# B&R Automation Studio project ChoiceBagging_SSBP (part 2)

#### Error.ld - Error detected
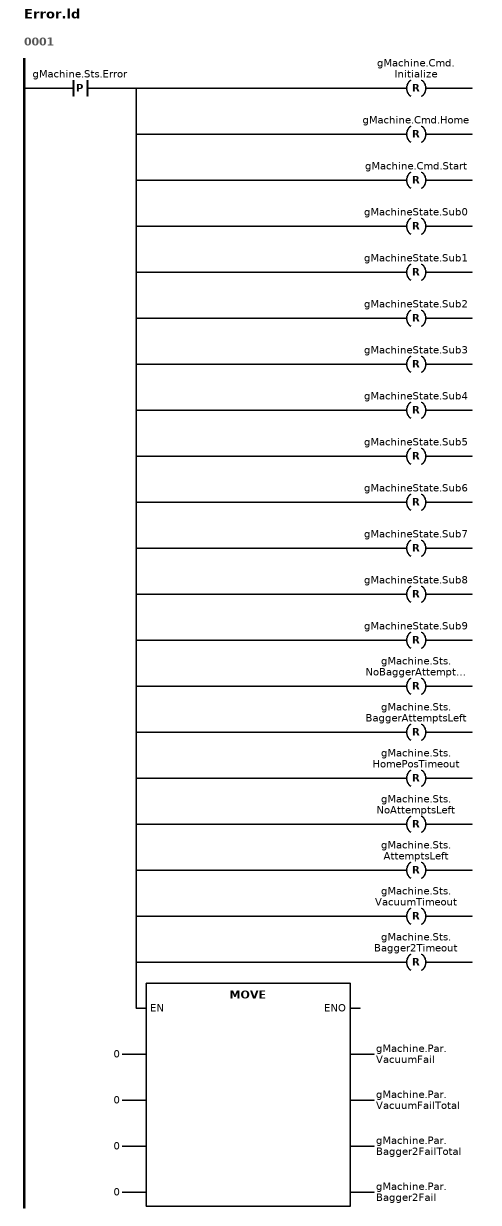
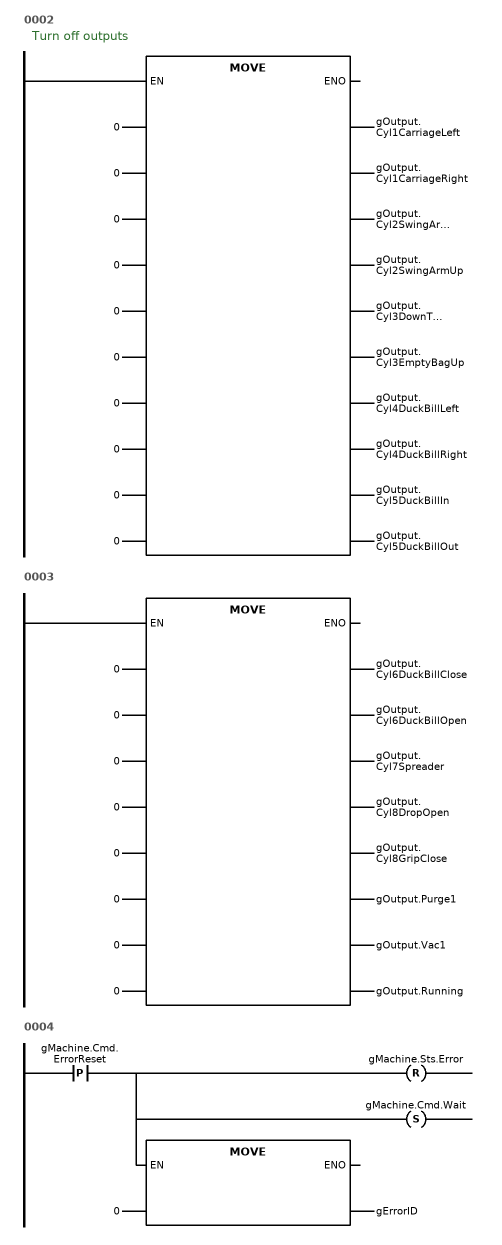
Ladder, written as Structured Text:
```iecst
ACTION Error:
VAR
    _e1 : R_TRIG;
    _e2 : R_TRIG;
END_VAR
(* Network 1 *)
_e1(CLK := gMachine.Sts.Error);
IF _e1.Q THEN
    gMachine.Cmd.Initialize := FALSE;
    gMachine.Cmd.Home := FALSE;
    gMachine.Cmd.Start := FALSE;
    gMachineState.Sub0 := FALSE;
    gMachineState.Sub1 := FALSE;
    gMachineState.Sub2 := FALSE;
    gMachineState.Sub3 := FALSE;
    gMachineState.Sub4 := FALSE;
    gMachineState.Sub5 := FALSE;
    gMachineState.Sub6 := FALSE;
    gMachineState.Sub7 := FALSE;
    gMachineState.Sub8 := FALSE;
    gMachineState.Sub9 := FALSE;
    gMachine.Sts.NoBaggerAttemptsLeft := FALSE;
    gMachine.Sts.BaggerAttemptsLeft := FALSE;
    gMachine.Sts.HomePosTimeout := FALSE;
    gMachine.Sts.NoAttemptsLeft := FALSE;
    gMachine.Sts.AttemptsLeft := FALSE;
    gMachine.Sts.VacuumTimeout := FALSE;
    gMachine.Sts.Bagger2Timeout := FALSE;
    gMachine.Par.VacuumFail := 0;
    gMachine.Par.VacuumFailTotal := 0;
    gMachine.Par.Bagger2FailTotal := 0;
    gMachine.Par.Bagger2Fail := 0;
END_IF;

(* Network 2: Turn off outputs *)
gOutput.Cyl1CarriageLeft := 0;
gOutput.Cyl1CarriageRight := 0;
gOutput.Cyl2SwingArmDown := 0;
gOutput.Cyl2SwingArmUp := 0;
gOutput.Cyl3DownToEmptyBag := 0;
gOutput.Cyl3EmptyBagUp := 0;
gOutput.Cyl4DuckBillLeft := 0;
gOutput.Cyl4DuckBillRight := 0;
gOutput.Cyl5DuckBillIn := 0;
gOutput.Cyl5DuckBillOut := 0;

(* Network 3 *)
gOutput.Cyl6DuckBillClose := 0;
gOutput.Cyl6DuckBillOpen := 0;
gOutput.Cyl7Spreader := 0;
gOutput.Cyl8DropOpen := 0;
gOutput.Cyl8GripClose := 0;
gOutput.Purge1 := 0;
gOutput.Vac1 := 0;
gOutput.Running := 0;

(* Network 4 *)
_e2(CLK := gMachine.Cmd.ErrorReset);
IF _e2.Q THEN
    gMachine.Sts.Error := FALSE;
    gMachine.Cmd.Wait := TRUE;
    gErrorID := 0;
END_IF;
END_ACTION
```

#### Wait.ld -  Waiting
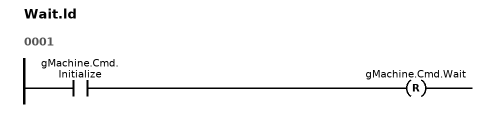
Ladder, written as Structured Text:
```iecst
ACTION Wait:
(* Network 1 *)
IF gMachine.Cmd.Initialize THEN gMachine.Cmd.Wait := FALSE; END_IF;
END_ACTION
```

#### Pause.ld - Pause / resume
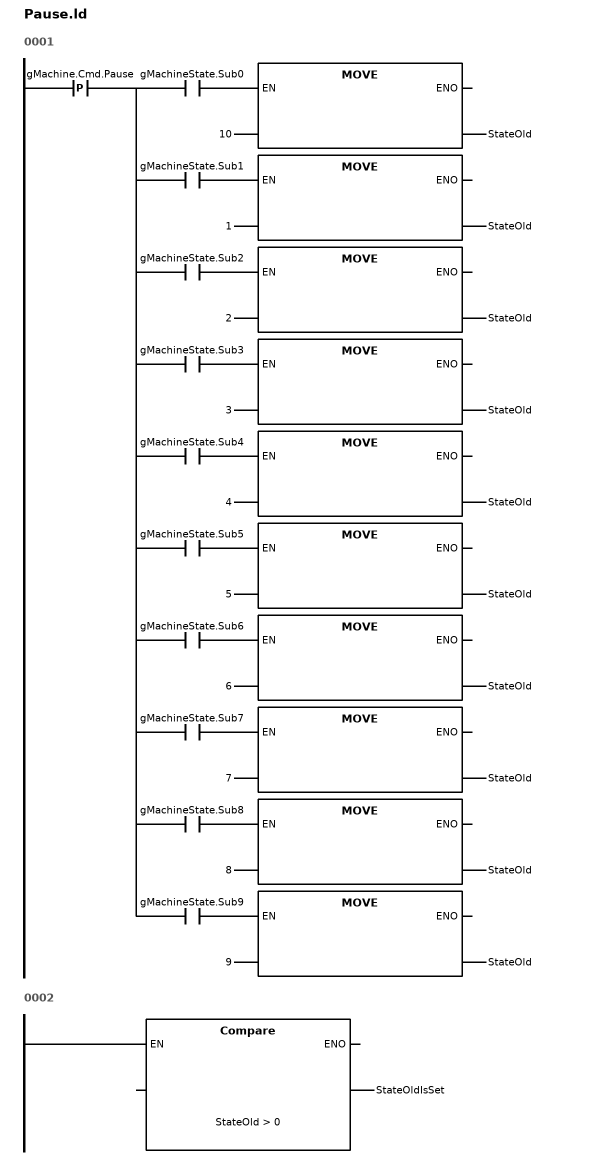
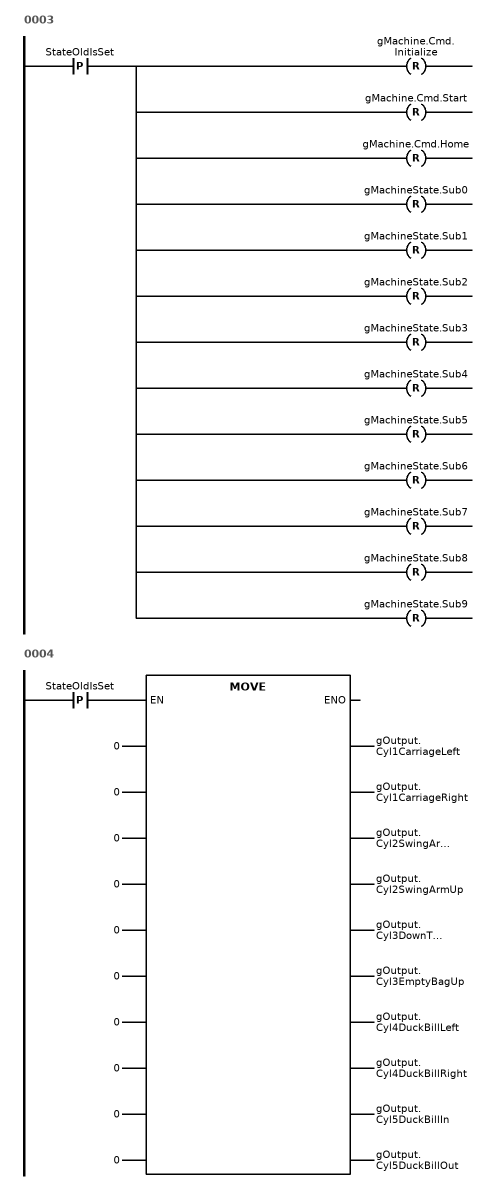
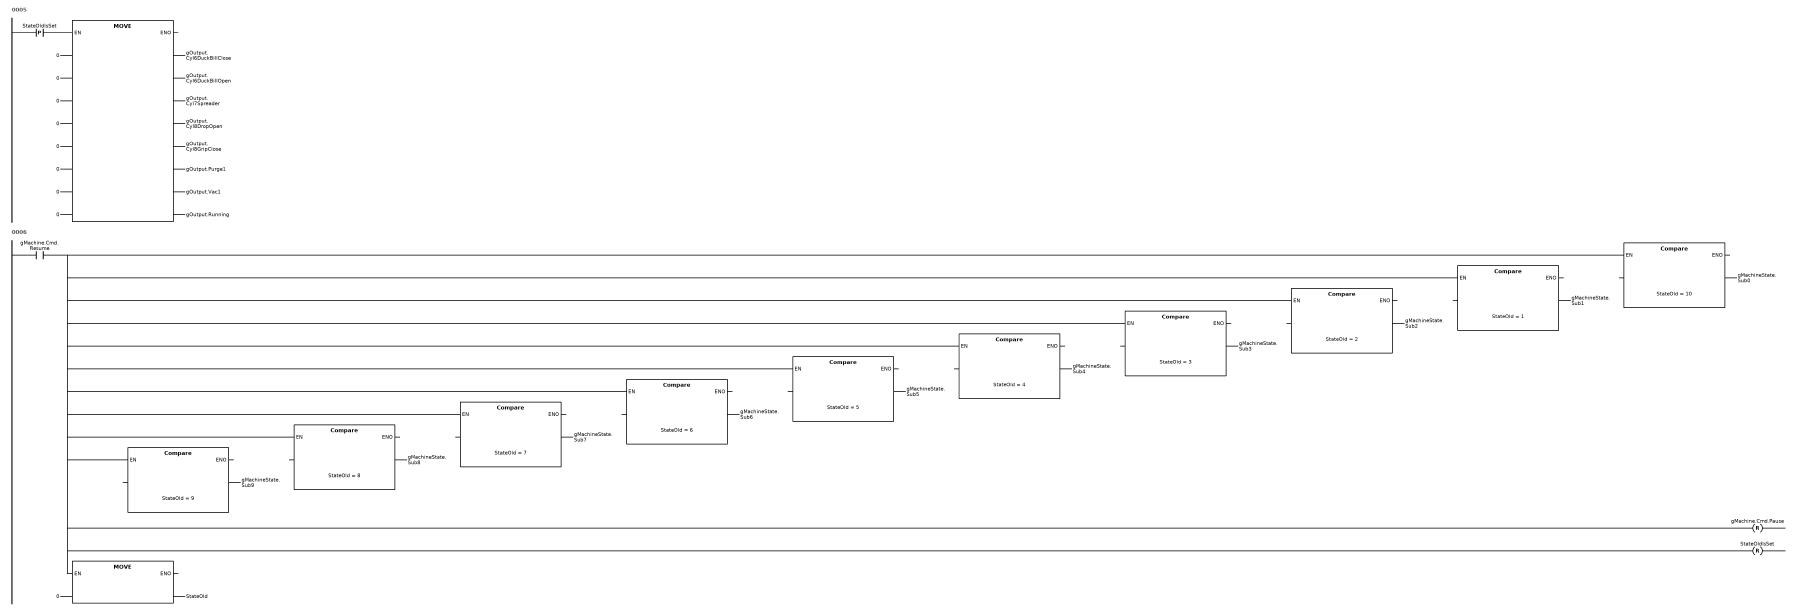
Ladder, written as Structured Text:
```iecst
ACTION Pause:
VAR
    _e1 : R_TRIG;
    _e2 : R_TRIG;
    _e3 : R_TRIG;
    _e4 : R_TRIG;
    _p5 : BOOL;
END_VAR
(* Network 1 *)
_e1(CLK := gMachine.Cmd.Pause);
IF _e1.Q AND gMachineState.Sub0 THEN StateOld := 10; END_IF;
IF _e1.Q AND gMachineState.Sub1 THEN StateOld := 1; END_IF;
IF _e1.Q AND gMachineState.Sub2 THEN StateOld := 2; END_IF;
IF _e1.Q AND gMachineState.Sub3 THEN StateOld := 3; END_IF;
IF _e1.Q AND gMachineState.Sub4 THEN StateOld := 4; END_IF;
IF _e1.Q AND gMachineState.Sub5 THEN StateOld := 5; END_IF;
IF _e1.Q AND gMachineState.Sub6 THEN StateOld := 6; END_IF;
IF _e1.Q AND gMachineState.Sub7 THEN StateOld := 7; END_IF;
IF _e1.Q AND gMachineState.Sub8 THEN StateOld := 8; END_IF;
IF _e1.Q AND gMachineState.Sub9 THEN StateOld := 9; END_IF;

(* Network 2 *)
StateOldIsSet := StateOld > 0;

(* Network 3 *)
_e2(CLK := StateOldIsSet);
IF _e2.Q THEN
    gMachine.Cmd.Initialize := FALSE;
    gMachine.Cmd.Start := FALSE;
    gMachine.Cmd.Home := FALSE;
    gMachineState.Sub0 := FALSE;
    gMachineState.Sub1 := FALSE;
    gMachineState.Sub2 := FALSE;
    gMachineState.Sub3 := FALSE;
    gMachineState.Sub4 := FALSE;
    gMachineState.Sub5 := FALSE;
    gMachineState.Sub6 := FALSE;
    gMachineState.Sub7 := FALSE;
    gMachineState.Sub8 := FALSE;
    gMachineState.Sub9 := FALSE;
END_IF;

(* Network 4 *)
_e3(CLK := StateOldIsSet);
IF _e3.Q THEN
    gOutput.Cyl1CarriageLeft := 0;
    gOutput.Cyl1CarriageRight := 0;
    gOutput.Cyl2SwingArmDown := 0;
    gOutput.Cyl2SwingArmUp := 0;
    gOutput.Cyl3DownToEmptyBag := 0;
    gOutput.Cyl3EmptyBagUp := 0;
    gOutput.Cyl4DuckBillLeft := 0;
    gOutput.Cyl4DuckBillRight := 0;
    gOutput.Cyl5DuckBillIn := 0;
    gOutput.Cyl5DuckBillOut := 0;
END_IF;

(* Network 5 *)
_e4(CLK := StateOldIsSet);
IF _e4.Q THEN
    gOutput.Cyl6DuckBillClose := 0;
    gOutput.Cyl6DuckBillOpen := 0;
    gOutput.Cyl7Spreader := 0;
    gOutput.Cyl8DropOpen := 0;
    gOutput.Cyl8GripClose := 0;
    gOutput.Purge1 := 0;
    gOutput.Vac1 := 0;
    gOutput.Running := 0;
END_IF;

(* Network 6 *)
IF gMachine.Cmd.Resume THEN
    gMachineState.Sub0 := StateOld = 10;
    gMachineState.Sub1 := StateOld = 1;
    gMachineState.Sub2 := StateOld = 2;
    gMachineState.Sub3 := StateOld = 3;
    gMachineState.Sub4 := StateOld = 4;
    gMachineState.Sub5 := StateOld = 5;
    gMachineState.Sub6 := StateOld = 6;
    gMachineState.Sub7 := StateOld = 7;
    gMachineState.Sub8 := StateOld = 8;
    gMachineState.Sub9 := StateOld = 9;
END_IF;
_p5 := gMachine.Cmd.Resume;
IF gMachine.Cmd.Resume THEN gMachine.Cmd.Pause := FALSE; END_IF;
IF _p5 THEN
    StateOldIsSet := FALSE;
    StateOld := 0;
END_IF;
END_ACTION
```

### Program Logical/AlarmCtrl (IEC)

#### Cyclic.ld - Cyclic code
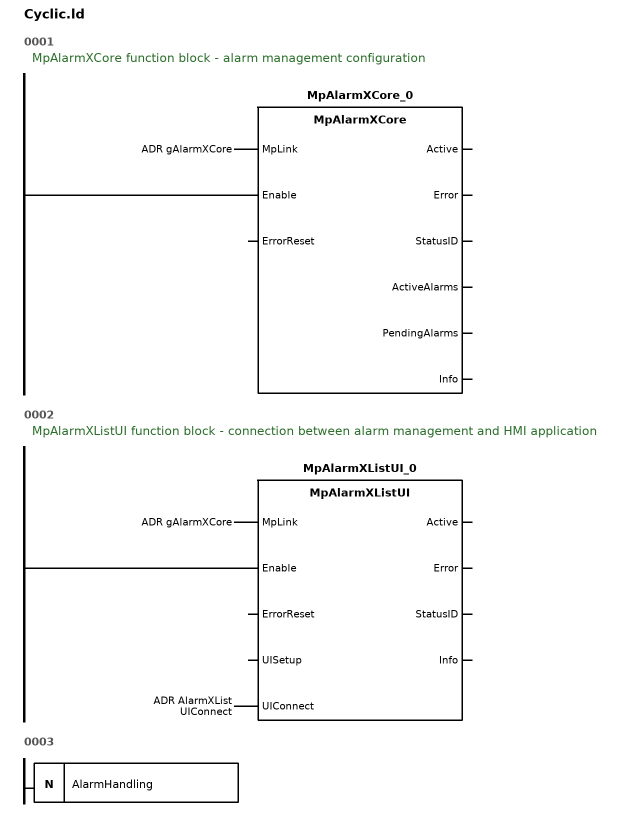
Ladder, written as Structured Text:
```iecst
(*********************************************************************************
 * Copyright: 	Hartfiel Automation
 * Author:    	cashley
 * Created:   	August 5, 2019/2:01 PM
 * Description: This file contains the control logic for handling the alarm system.
 *********************************************************************************)
 PROGRAM _CYCLIC
(* Network 1: MpAlarmXCore function block - alarm management configuration *)
MpAlarmXCore_0(MpLink := ADR(gAlarmXCore), Enable := TRUE);

(* Network 2: MpAlarmXListUI function block - connection between alarm management and HMI application *)
MpAlarmXListUI_0(MpLink := ADR(gAlarmXCore), Enable := TRUE, UIConnect := ADR(AlarmXListUIConnect));

(* Network 3 *)
AlarmHandling;
END_PROGRAM
```

#### Variables.var - Local variables
```iecst
VAR
	MpAlarmXCore_0 : MpAlarmXCore; (*Function block for MpAlarmXCore*)
	MpAlarmXListUI_0 : MpAlarmXListUI; (*Function block for MpAlarmXListUI*)
	AlarmXListUIConnect : MpAlarmXListUIConnectType; (*MpAlarmXListUIConnect type*)
	ErrorString : STRING[255]; (*String for MpAlarmXSet unique alarm code*)
END_VAR
```

#### AlarmHandling.st - Alarm handling
```iecst
ACTION AlarmHandling:

	//Error ID determines unique name for MpAlarmXSet
	IF gErrorID = HOMING_TIMEOUT THEN
		ErrorString := 'HomingTimeout';
	ELSIF gErrorID = SAFE_TO_RUN THEN
		ErrorString := 'SafetyStatus';
	ELSIF gErrorID = CONVEYOR THEN
		ErrorString := 'ConveyorStatus';
	ELSIF gErrorID = MODULE_OK THEN
		ErrorString := 'ModuleStatus';
	ELSIF gErrorID = VACUUM_FAILURE THEN
		ErrorString := 'VacuumFailure';
	ELSIF gErrorID = BAG_ON_SPOUT_FAILURE THEN
		ErrorString := 'Bagger2Failure';
	END_IF

	//MpAlarmXSet - enables user-defined alarms
	IF EDGEPOS(gMachine.Sts.Error) THEN
		MpAlarmXSet(MpLink := gAlarmXCore, Name := ErrorString);
	END_IF

	//Error acknowledge and reset
	IF gMachine.Sts.Error = FALSE THEN
		gMachine.Cmd.ErrorReset := FALSE;
	END_IF

END_ACTION
```

### Program Logical/IOCtrl (IEC)

#### Cyclic.ld
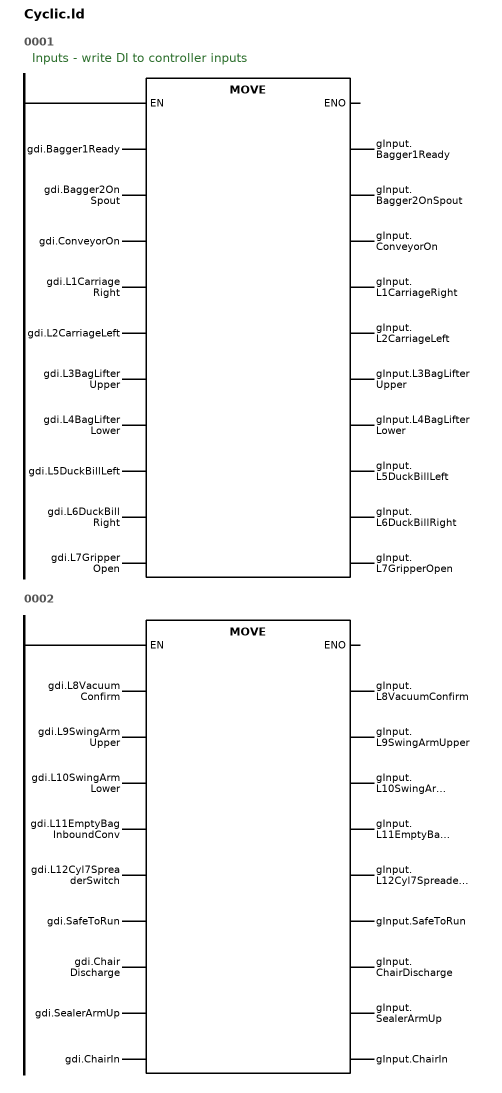
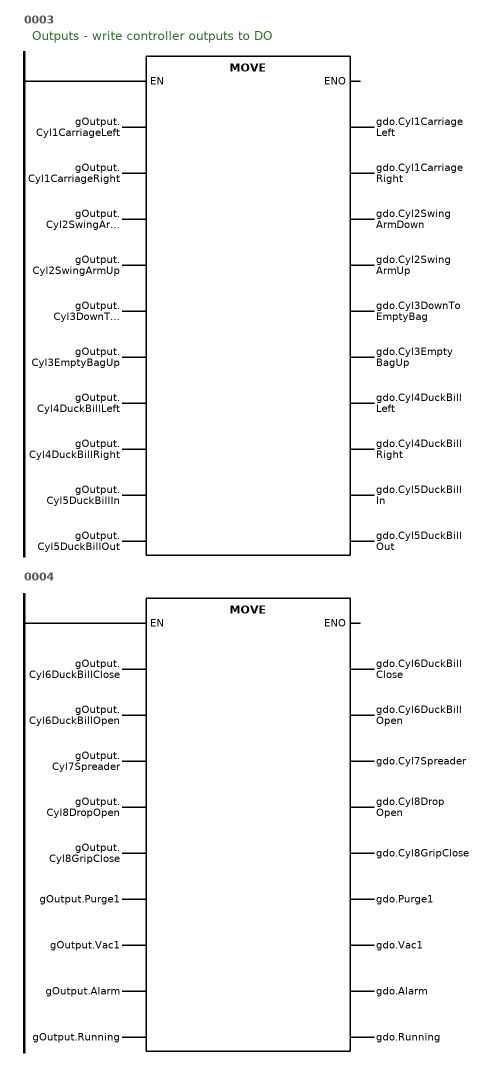
Ladder, written as Structured Text:
```iecst
(*********************************************************************************
 * Copyright: 	Hartfiel Automation
 * Author:    	cashley
 * Created:   	August 5, 2019/2:01 PM
 * Description: This file contains the control logic for the inputs and outputs.
 *********************************************************************************)
 PROGRAM _CYCLIC
(* Network 1: Inputs - write DI to controller inputs *)
gInput.Bagger1Ready := gdi.Bagger1Ready;
gInput.Bagger2OnSpout := gdi.Bagger2OnSpout;
gInput.ConveyorOn := gdi.ConveyorOn;
gInput.L1CarriageRight := gdi.L1CarriageRight;
gInput.L2CarriageLeft := gdi.L2CarriageLeft;
gInput.L3BagLifterUpper := gdi.L3BagLifterUpper;
gInput.L4BagLifterLower := gdi.L4BagLifterLower;
gInput.L5DuckBillLeft := gdi.L5DuckBillLeft;
gInput.L6DuckBillRight := gdi.L6DuckBillRight;
gInput.L7GripperOpen := gdi.L7GripperOpen;

(* Network 2 *)
gInput.L8VacuumConfirm := gdi.L8VacuumConfirm;
gInput.L9SwingArmUpper := gdi.L9SwingArmUpper;
gInput.L10SwingArmLower := gdi.L10SwingArmLower;
gInput.L11EmptyBagInboundConv := gdi.L11EmptyBagInboundConv;
gInput.L12Cyl7SpreaderSwitch := gdi.L12Cyl7SpreaderSwitch;
gInput.SafeToRun := gdi.SafeToRun;
gInput.ChairDischarge := gdi.ChairDischarge;
gInput.SealerArmUp := gdi.SealerArmUp;
gInput.ChairIn := gdi.ChairIn;

(* Network 3: Outputs - write controller outputs to DO *)
gdo.Cyl1CarriageLeft := gOutput.Cyl1CarriageLeft;
gdo.Cyl1CarriageRight := gOutput.Cyl1CarriageRight;
gdo.Cyl2SwingArmDown := gOutput.Cyl2SwingArmDown;
gdo.Cyl2SwingArmUp := gOutput.Cyl2SwingArmUp;
gdo.Cyl3DownToEmptyBag := gOutput.Cyl3DownToEmptyBag;
gdo.Cyl3EmptyBagUp := gOutput.Cyl3EmptyBagUp;
gdo.Cyl4DuckBillLeft := gOutput.Cyl4DuckBillLeft;
gdo.Cyl4DuckBillRight := gOutput.Cyl4DuckBillRight;
gdo.Cyl5DuckBillIn := gOutput.Cyl5DuckBillIn;
gdo.Cyl5DuckBillOut := gOutput.Cyl5DuckBillOut;

(* Network 4 *)
gdo.Cyl6DuckBillClose := gOutput.Cyl6DuckBillClose;
gdo.Cyl6DuckBillOpen := gOutput.Cyl6DuckBillOpen;
gdo.Cyl7Spreader := gOutput.Cyl7Spreader;
gdo.Cyl8DropOpen := gOutput.Cyl8DropOpen;
gdo.Cyl8GripClose := gOutput.Cyl8GripClose;
gdo.Purge1 := gOutput.Purge1;
gdo.Vac1 := gOutput.Vac1;
gdo.Alarm := gOutput.Alarm;
gdo.Running := gOutput.Running;
END_PROGRAM
```

#### Init.ld
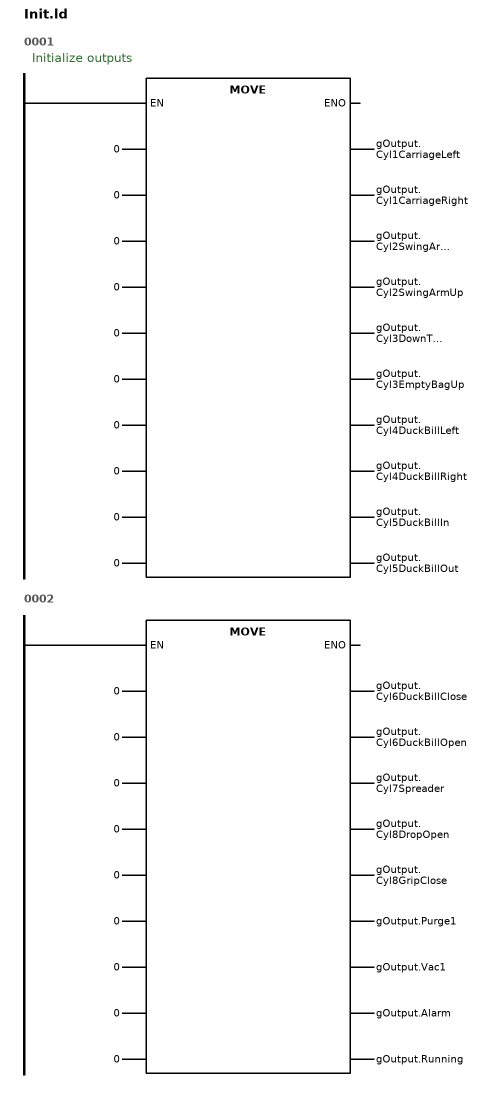
Ladder, written as Structured Text:
```iecst
PROGRAM _INIT
(* Network 1: Initialize outputs *)
gOutput.Cyl1CarriageLeft := 0;
gOutput.Cyl1CarriageRight := 0;
gOutput.Cyl2SwingArmDown := 0;
gOutput.Cyl2SwingArmUp := 0;
gOutput.Cyl3DownToEmptyBag := 0;
gOutput.Cyl3EmptyBagUp := 0;
gOutput.Cyl4DuckBillLeft := 0;
gOutput.Cyl4DuckBillRight := 0;
gOutput.Cyl5DuckBillIn := 0;
gOutput.Cyl5DuckBillOut := 0;

(* Network 2 *)
gOutput.Cyl6DuckBillClose := 0;
gOutput.Cyl6DuckBillOpen := 0;
gOutput.Cyl7Spreader := 0;
gOutput.Cyl8DropOpen := 0;
gOutput.Cyl8GripClose := 0;
gOutput.Purge1 := 0;
gOutput.Vac1 := 0;
gOutput.Alarm := 0;
gOutput.Running := 0;
END_PROGRAM
```

- Visualisation Logical/Visualization (not shown)

Listed in the project but not available here: Logical/MainCtrl/Exit.ld, Logical/MainCtrl/Types.typ, Logical/AlarmCtrl/Init.ld, Logical/AlarmCtrl/Exit.ld, Logical/AlarmCtrl/Types.typ
